(* IEC 61131-3 sources: AXOpen/src/abstractions/ctrl/src/Messaging, 18 files *)

(* ---- AxoConstants.st ---- *)
NAMESPACE AXOpen.Messaging
    TYPE PUBLIC
        AxoIntConstants : INT
        (
            MAX_MESSAGE_TEXT_LENGHT := 160,
			MDS_MAX_INDEX := 10
        );
    END_TYPE
END_NAMESPACE

(* ---- eAxoMessageDigestMethod.st ---- *)
NAMESPACE AXOpen.Messaging
    /// <summary>
    /// Message digest methods used to create fingerprint of a message.
    /// </summary>
    TYPE eAxoMessageDigestMethod : INT
    (
        /// <summary>
        /// Fastest method with highest probability of colisions.
        /// </summary>
        CRC8 := 8,

        /// <summary>
        /// Moderate speed method with lower probability of colisions.
        /// </summary>
        CRC16 := 16,

        /// <summary>
        /// Slowest speed method with relatively low probability of colisions.
        /// </summary>
        CRC32 := 32,

        /// <summary>
        /// Messages are not digested the repeated messages won't be filtered out.
        /// Use this option on low performance devices.
        /// </summary>
        NONE := 32767
    );
    END_TYPE
END_NAMESPACE

(* ---- IAxoMessageCategorize.st ---- *)
NAMESPACE AXOpen.Messaging
    INTERFACE IAxoMessageCategorize
		/// <summary>
        /// Categorizes and creates the message as 'debug'.
		/// </summary>
        METHOD AsDebug : IAxoMessageProperties END_METHOD

		/// <summary>
        /// Categorizes and creates the message as 'error'.
		/// </summary>
        METHOD AsError : IAxoMessageProperties END_METHOD

		/// <summary>
        /// Categorizes and creates the message as 'fatal'.
		/// </summary>
        METHOD AsFatal : IAxoMessageProperties END_METHOD

		/// <summary>
        /// Categorizes and creates the message as 'info'.
		/// </summary>
        METHOD AsInfo : IAxoMessageProperties END_METHOD

		/// <summary>
        /// Categorizes and creates the message as 'trace'.
		/// </summary>
        METHOD AsTrace : IAxoMessageProperties END_METHOD

		/// <summary>
        /// Categorizes and creates the message as 'warning'.
		/// </summary>
        METHOD AsWarning : IAxoMessageProperties END_METHOD
    END_INTERFACE
END_NAMESPACE

(* ---- IAxoMessageProperties.st ---- *)
NAMESPACE AXOpen.Messaging
    INTERFACE IAxoMessageProperties
        METHOD Pin: IAxoMessageProperties END_METHOD
        METHOD IsPinned: BOOL END_METHOD
    END_INTERFACE
END_NAMESPACE

(* ---- IAxoMessages.st ---- *)
NAMESPACE AXOpen.Messaging
    INTERFACE IAxoMessages
	    /// <summary>
		/// Adds message of 'debug' category to the message queue.
		/// </summary>
        METHOD Debug : IAxoMessageProperties
            VAR_INPUT
                /// <summary>
                /// Arbitrary message string.
                /// </summary>
                Message : STRING[AxoIntConstants#MAX_MESSAGE_TEXT_LENGHT];
            END_VAR
        END_METHOD

	    /// <summary>
		/// Adds message of 'error' category to the message queue.
		/// </summary>
        METHOD Error : IAxoMessageProperties
            VAR_INPUT
                /// <summary>
                /// Arbitrary message string.
                /// </summary>
                Message : STRING[AxoIntConstants#MAX_MESSAGE_TEXT_LENGHT];
            END_VAR
        END_METHOD

	    /// <summary>
		/// Adds message of 'information' category to the message queue.
		/// </summary>
        METHOD Info : IAxoMessageProperties
            VAR_INPUT
                /// <summary>
                /// Arbitrary message string.
                /// </summary>
                Message : STRING[AxoIntConstants#MAX_MESSAGE_TEXT_LENGHT];
            END_VAR
        END_METHOD

	    /// <summary>
		/// Adds message of 'notification' category to the message queue.
		/// </summary>
        METHOD Notify : IAxoMessageProperties
            VAR_INPUT
                /// <summary>
                /// Arbitrary message string.
                /// </summary>
                Message : STRING[AxoIntConstants#MAX_MESSAGE_TEXT_LENGHT];
            END_VAR
        END_METHOD

	    /// <summary>
		/// Adds message of 'programming error' category to the message queue.
		/// </summary>
        METHOD Programming : IAxoMessageProperties
            VAR_INPUT
                /// <summary>
                /// Arbitrary message string.
                /// </summary>
                Message : STRING[AxoIntConstants#MAX_MESSAGE_TEXT_LENGHT];
            END_VAR
        END_METHOD

	    /// <summary>
		/// Adds message of 'trace' category to the message queue.
		/// </summary>
        METHOD Trace : IAxoMessageProperties
            VAR_INPUT
                /// <summary>
                /// Arbitrary message string.
                /// </summary>
                Message : STRING[AxoIntConstants#MAX_MESSAGE_TEXT_LENGHT];
            END_VAR
        END_METHOD

	    /// <summary>
		/// Adds message of 'warning' category to the message queue.
		/// </summary>
        METHOD Warning : IAxoMessageProperties
            VAR_INPUT
                /// <summary>
                /// Arbitrary message string.
                /// </summary>
                Message : STRING[AxoIntConstants#MAX_MESSAGE_TEXT_LENGHT];
            END_VAR
        END_METHOD

        METHOD Build: IAxoMessageTextBuilder END_METHOD

        /// <summary>
		/// Adds message of given category to the message queue.
		/// </summary>
		/// <returns>Message index.</returns>
        METHOD Post  : IAxoMessageProperties
            VAR_INPUT
                /// <summary>
                /// Arbitrary message string.
                /// </summary>
                Message : STRING[AxoIntConstants#MAX_MESSAGE_TEXT_LENGHT];
                /// <summary>
                /// Message category.
                /// </summary>
                Category : eAxoMessageCategory;
            END_VAR
        END_METHOD

		/// <summary>
		/// Unpins this messenger.
		/// </summary>
        METHOD UnPin END_METHOD

    END_INTERFACE
END_NAMESPACE

(* ---- IAxoMessageTextBuilder.st ---- *)
NAMESPACE AXOpen.Messaging
    INTERFACE IAxoMessageTextBuilder
		/// <summary>
		/// Appends string to the message text.
		/// </summary>
		/// <remarks>
		/// 	<note type="warning">
		/// 		The size of the resulting string should not be more than '160' characters. The characters exceeding this size will be truncated.
		/// 	</note>
		/// </remarks>
 		METHOD Append : IAxoMessageTextBuilder VAR_INPUT Data : BOOL; END_VAR END_METHOD
		METHOD Append : IAxoMessageTextBuilder VAR_INPUT Data : BYTE; END_VAR END_METHOD
		METHOD Append : IAxoMessageTextBuilder VAR_INPUT Data : WORD; END_VAR END_METHOD
		METHOD Append : IAxoMessageTextBuilder VAR_INPUT Data : DWORD; END_VAR END_METHOD
		METHOD Append : IAxoMessageTextBuilder VAR_INPUT Data : LWORD; END_VAR END_METHOD
		METHOD Append : IAxoMessageTextBuilder VAR_INPUT Data : SINT; END_VAR END_METHOD
		METHOD Append : IAxoMessageTextBuilder VAR_INPUT Data : INT; END_VAR END_METHOD
		METHOD Append : IAxoMessageTextBuilder VAR_INPUT Data : DINT; END_VAR END_METHOD
		METHOD Append : IAxoMessageTextBuilder VAR_INPUT Data : LINT; END_VAR END_METHOD
		METHOD Append : IAxoMessageTextBuilder VAR_INPUT Data : USINT; END_VAR END_METHOD
		METHOD Append : IAxoMessageTextBuilder VAR_INPUT Data : UINT; END_VAR END_METHOD
		METHOD Append : IAxoMessageTextBuilder VAR_INPUT Data : UDINT; END_VAR END_METHOD
		METHOD Append : IAxoMessageTextBuilder VAR_INPUT Data : ULINT; END_VAR END_METHOD
		METHOD Append : IAxoMessageTextBuilder VAR_INPUT Data : REAL; END_VAR END_METHOD
		METHOD Append : IAxoMessageTextBuilder VAR_INPUT Data : LREAL; END_VAR END_METHOD
		METHOD Append : IAxoMessageTextBuilder VAR_INPUT Data : TIME; END_VAR END_METHOD
		METHOD Append : IAxoMessageTextBuilder VAR_INPUT Data : LTIME; END_VAR END_METHOD
		METHOD Append : IAxoMessageTextBuilder VAR_INPUT Data : DATE; END_VAR END_METHOD
		METHOD Append : IAxoMessageTextBuilder VAR_INPUT Data : LDATE; END_VAR END_METHOD
		METHOD Append : IAxoMessageTextBuilder VAR_INPUT Data : TIME_OF_DAY; END_VAR END_METHOD
		METHOD Append : IAxoMessageTextBuilder VAR_INPUT Data : LTIME_OF_DAY; END_VAR END_METHOD
		METHOD Append : IAxoMessageTextBuilder VAR_INPUT Data : DATE_AND_TIME; END_VAR END_METHOD
		METHOD Append : IAxoMessageTextBuilder VAR_INPUT Data : LDATE_AND_TIME; END_VAR END_METHOD
		METHOD Append : IAxoMessageTextBuilder VAR_INPUT Data : CHAR; END_VAR END_METHOD
		// METHOD Append : IAxoMessageTextBuilder VAR_INPUT Data : WCHAR; END_VAR END_METHOD
		METHOD Append : IAxoMessageTextBuilder VAR_INPUT Data : STRING[AxoIntConstants#MAX_MESSAGE_TEXT_LENGHT]; END_VAR END_METHOD
		// METHOD Append : IAxoMessageTextBuilder VAR_INPUT Data : WSTRING[IxIntConstants#MAX_MESSAGE_TEXT_LENGHT]; END_VAR END_METHOD
		/// <summary>
		/// Gets categorization methods for fluent message builder.
		/// </summary>
        METHOD As : IAxoMessageCategorize END_METHOD

		/// <summary>
		/// Initiates new message text building for this messenger in fluent-like fashion.
		/// </summary>
        METHOD Build : IAxoMessageTextBuilder END_METHOD
    END_INTERFACE
END_NAMESPACE

(* ---- IAxoMessenger.st ---- *)
NAMESPACE AXOpen.Messaging
    INTERFACE IAxoMessenger
		/// <summary>
		/// Clears the message content.
		/// <remarks>
		/// 	<note type="important">
		/// 		This method is exposed for Rpc calls, for testing purposes. Rpc calls of this method must not be used in production code
		///		</note>
		/// </remarks>
		/// </summary>
		METHOD Clear END_METHOD

		METHOD OnCondition : IAxoMessages
			VAR_INPUT
				inCondition : BOOL;
			END_VAR
		END_METHOD
    END_INTERFACE
END_NAMESPACE

(* ---- IAxoMessengerEnv.st ---- *)
NAMESPACE AXOpen.Messaging
    INTERFACE IAxoMessengerEnv
		/// <summary>
		/// Gets whether the messaging is suspended at this point in program.
		/// <para>
		/// See also <see cref="PlcDocu.TcoCore.TcoMessengerSettings.Resume()"/>
		/// </para>
		/// <para>
		/// See also <see cref="PlcDocu.TcoCore.TcoMessengerSettings.Suspend()"/>
		/// </para>
		/// <para>
		/// See also <see cref="PlcDocu.TcoCore.TcoMessengerSettings.MinLevel"/>
		/// </para>
		/// </summary>
		METHOD IsSuspended: BOOL END_METHOD
		/// <summary>
		/// Gets the message digest method.
		/// Message digest serves to fingerprint messages.
		/// </summary>
		METHOD GetMessageDigestMethod : eAxoMessageDigestMethod END_METHOD
		/// <summary>
		/// Sets the message digest method.
		/// Message digest serves to fingerprint messages.
		/// </summary>
		METHOD SetMessageDigestMethod VAR_INPUT inDigestMethod : eAxoMessageDigestMethod; END_VAR END_METHOD
		/// <summary>
		/// Gets the minimal messaging level, the objects will post only messages for the levels of this or superior severity.
		/// <para>
		/// See also <see cref="PlcDocu.TcoCore.TcoMessengerSettings.Resume()"/>
		/// </para>
		/// <para>
		/// See also <see cref="PlcDocu.TcoCore.TcoMessengerSettings.Suspend()"/>
		/// </para>
		/// <para>
		/// See also <see cref="PlcDocu.TcoCore.TcoMessengerSettings.MinLevel"/>
		/// </para>
		/// </summary>
		METHOD GetMinLevel : eAxoMessageCategory END_METHOD
		/// <summary>
		/// Sets the minimal messaging level, the objects will post only messages for the levels of this or superior severity.
		/// <para>
		/// See also <see cref="PlcDocu.TcoCore.TcoMessengerSettings.Resume()"/>
		/// </para>
		/// <para>
		/// See also <see cref="PlcDocu.TcoCore.TcoMessengerSettings.Suspend()"/>
		/// </para>
		/// <para>
		/// See also <see cref="PlcDocu.TcoCore.TcoMessengerSettings.MinLevel"/>
		/// </para>
		/// </summary>
		METHOD SetMinLevel VAR_INPUT inMessageCategory : eAxoMessageCategory; END_VAR END_METHOD
		/// <summary>
		/// Resumes messaging from the all objects of this context, when the messaging was previously suspended by ```Suspend``` method.
		/// <para>
		/// See also <see cref="PlcDocu.TcoCore.TcoMessengerSettings.Suspend()"/>
		/// </para>
		/// <para>
		/// See also <see cref="PlcDocu.TcoCore.TcoMessengerSettings.MinLevel"/>
		/// </para>
		/// </summary>
		METHOD Resume END_METHOD
		/// <summary>
		/// Suspends messaging from the all objects of this context that would occur from this point in the call tree.
		/// <para>
		/// See also <see cref="PlcDocu.TcoCore.TcoMessengerSettings.Resume()"/>
		/// </para>
		/// <para>
		/// See also <see cref="PlcDocu.TcoCore.TcoMessengerSettings.MinLevel"/>
		/// </para>
		/// </summary>
		METHOD Suspend END_METHOD
	END_INTERFACE
END_NAMESPACE

(* ---- IIxMessageCategorize.st ---- *)
NAMESPACE ix.framework.messaging
    INTERFACE IIxMessageCategorize
		/// <summary>
        /// Categorizes and creates the message as 'debug'.
		/// </summary>
        METHOD AsDebug : IIxMessageProperties END_METHOD

		/// <summary>
        /// Categorizes and creates the message as 'error'.
		/// </summary>
        METHOD AsError : IIxMessageProperties END_METHOD

		/// <summary>
        /// Categorizes and creates the message as 'fatal'.
		/// </summary>
        METHOD AsFatal : IIxMessageProperties END_METHOD

		/// <summary>
        /// Categorizes and creates the message as 'info'.
		/// </summary>
        METHOD AsInfo : IIxMessageProperties END_METHOD

		/// <summary>
        /// Categorizes and creates the message as 'trace'.
		/// </summary>
        METHOD AsTrace : IIxMessageProperties END_METHOD

		/// <summary>
        /// Categorizes and creates the message as 'warning'.
		/// </summary>
        METHOD AsWarning : IIxMessageProperties END_METHOD
    END_INTERFACE
END_NAMESPACE

(* ---- IIxMessages.st ---- *)
NAMESPACE ix.framework.messaging
    INTERFACE IIxMessages
	    /// <summary>
		/// Adds message of 'debug' category to the message queue.
		/// </summary>
        METHOD Debug : IIxMessageProperties
            VAR_INPUT
                /// <summary>
                /// Arbitrary message string.
                /// </summary>
                Message : STRING[IxIntConstants#MAX_MESSAGE_TEXT_LENGHT];
            END_VAR
        END_METHOD

	    /// <summary>
		/// Adds message of 'error' category to the message queue.
		/// </summary>
        METHOD Error : IIxMessageProperties
            VAR_INPUT
                /// <summary>
                /// Arbitrary message string.
                /// </summary>
                Message : STRING[IxIntConstants#MAX_MESSAGE_TEXT_LENGHT];
            END_VAR
        END_METHOD

	    /// <summary>
		/// Adds message of 'information' category to the message queue.
		/// </summary>
        METHOD Info : IIxMessageProperties
            VAR_INPUT
                /// <summary>
                /// Arbitrary message string.
                /// </summary>
                Message : STRING[IxIntConstants#MAX_MESSAGE_TEXT_LENGHT];
            END_VAR
        END_METHOD

	    /// <summary>
		/// Adds message of 'notification' category to the message queue.
		/// </summary>
        METHOD Notify : IIxMessageProperties
            VAR_INPUT
                /// <summary>
                /// Arbitrary message string.
                /// </summary>
                Message : STRING[IxIntConstants#MAX_MESSAGE_TEXT_LENGHT];
            END_VAR
        END_METHOD

	    /// <summary>
		/// Adds message of 'programming error' category to the message queue.
		/// </summary>
        METHOD Programming : IIxMessageProperties
            VAR_INPUT
                /// <summary>
                /// Arbitrary message string.
                /// </summary>
                Message : STRING[IxIntConstants#MAX_MESSAGE_TEXT_LENGHT];
            END_VAR
        END_METHOD

	    /// <summary>
		/// Adds message of 'trace' category to the message queue.
		/// </summary>
        METHOD Trace : IIxMessageProperties
            VAR_INPUT
                /// <summary>
                /// Arbitrary message string.
                /// </summary>
                Message : STRING[IxIntConstants#MAX_MESSAGE_TEXT_LENGHT];
            END_VAR
        END_METHOD

	    /// <summary>
		/// Adds message of 'warning' category to the message queue.
		/// </summary>
        METHOD Warning : IIxMessageProperties
            VAR_INPUT
                /// <summary>
                /// Arbitrary message string.
                /// </summary>
                Message : STRING[IxIntConstants#MAX_MESSAGE_TEXT_LENGHT];
            END_VAR
        END_METHOD

        METHOD Build: IIxMessageTextBuilder END_METHOD

        /// <summary>
		/// Adds message of given category to the message queue.
		/// </summary>
		/// <returns>Message index.</returns>
        METHOD Post  : IIxMessageProperties
            VAR_INPUT
                /// <summary>
                /// Arbitrary message string.
                /// </summary>
                Message : STRING[IxIntConstants#MAX_MESSAGE_TEXT_LENGHT];
                /// <summary>
                /// Message category.
                /// </summary>
                Category : eIxMessageCategory;
            END_VAR
        END_METHOD

		/// <summary>
		/// Unpins this messenger.
		/// </summary>
        METHOD UnPin END_METHOD

    END_INTERFACE
END_NAMESPACE

(* ---- IIxMessageTextBuilder.st ---- *)
NAMESPACE ix.framework.messaging
    INTERFACE IIxMessageTextBuilder
		/// <summary>
		/// Appends string to the message text.
		/// </summary>
		/// <remarks>
		/// 	<note type="warning">
		/// 		The size of the resulting string should not be more than '160' characters. The characters exceeding this size will be truncated.
		/// 	</note>
		/// </remarks>
 		METHOD Append : IIxMessageTextBuilder VAR_INPUT Data : BOOL; END_VAR END_METHOD
		METHOD Append : IIxMessageTextBuilder VAR_INPUT Data : BYTE; END_VAR END_METHOD
		METHOD Append : IIxMessageTextBuilder VAR_INPUT Data : WORD; END_VAR END_METHOD
		METHOD Append : IIxMessageTextBuilder VAR_INPUT Data : DWORD; END_VAR END_METHOD
		METHOD Append : IIxMessageTextBuilder VAR_INPUT Data : LWORD; END_VAR END_METHOD
		METHOD Append : IIxMessageTextBuilder VAR_INPUT Data : SINT; END_VAR END_METHOD
		METHOD Append : IIxMessageTextBuilder VAR_INPUT Data : INT; END_VAR END_METHOD
		METHOD Append : IIxMessageTextBuilder VAR_INPUT Data : DINT; END_VAR END_METHOD
		METHOD Append : IIxMessageTextBuilder VAR_INPUT Data : LINT; END_VAR END_METHOD
		METHOD Append : IIxMessageTextBuilder VAR_INPUT Data : USINT; END_VAR END_METHOD
		METHOD Append : IIxMessageTextBuilder VAR_INPUT Data : UINT; END_VAR END_METHOD
		METHOD Append : IIxMessageTextBuilder VAR_INPUT Data : UDINT; END_VAR END_METHOD
		METHOD Append : IIxMessageTextBuilder VAR_INPUT Data : ULINT; END_VAR END_METHOD
		METHOD Append : IIxMessageTextBuilder VAR_INPUT Data : REAL; END_VAR END_METHOD
		METHOD Append : IIxMessageTextBuilder VAR_INPUT Data : LREAL; END_VAR END_METHOD
		METHOD Append : IIxMessageTextBuilder VAR_INPUT Data : TIME; END_VAR END_METHOD
		METHOD Append : IIxMessageTextBuilder VAR_INPUT Data : LTIME; END_VAR END_METHOD
		METHOD Append : IIxMessageTextBuilder VAR_INPUT Data : DATE; END_VAR END_METHOD
		METHOD Append : IIxMessageTextBuilder VAR_INPUT Data : LDATE; END_VAR END_METHOD
		METHOD Append : IIxMessageTextBuilder VAR_INPUT Data : TIME_OF_DAY; END_VAR END_METHOD
		METHOD Append : IIxMessageTextBuilder VAR_INPUT Data : LTIME_OF_DAY; END_VAR END_METHOD
		METHOD Append : IIxMessageTextBuilder VAR_INPUT Data : DATE_AND_TIME; END_VAR END_METHOD
		METHOD Append : IIxMessageTextBuilder VAR_INPUT Data : LDATE_AND_TIME; END_VAR END_METHOD
		METHOD Append : IIxMessageTextBuilder VAR_INPUT Data : CHAR; END_VAR END_METHOD
		// METHOD Append : IIxMessageTextBuilder VAR_INPUT Data : WCHAR; END_VAR END_METHOD
		METHOD Append : IIxMessageTextBuilder VAR_INPUT Data : STRING[IxIntConstants#MAX_MESSAGE_TEXT_LENGHT]; END_VAR END_METHOD
		// METHOD Append : IIxMessageTextBuilder VAR_INPUT Data : WSTRING[IxIntConstants#MAX_MESSAGE_TEXT_LENGHT]; END_VAR END_METHOD
		/// <summary>
		/// Gets categorization methods for fluent message builder.
		/// </summary>
        METHOD As : IIxMessageCategorize END_METHOD

		/// <summary>
		/// Initiates new message text building for this messenger in fluent-like fashion.
		/// </summary>
        METHOD Build : IIxMessageTextBuilder END_METHOD
    END_INTERFACE
END_NAMESPACE

(* ---- IIxMessenger.st ---- *)
NAMESPACE ix.framework.messaging
    INTERFACE IIxMessenger
		/// <summary>
		/// Clears the message content.
		/// <remarks>
		/// 	<note type="important">
		/// 		This method is exposed for Rpc calls, for testing purposes. Rpc calls of this method must not be used in production code
		///		</note>
		/// </remarks>
		/// </summary>
		METHOD Clear END_METHOD

		METHOD OnCondition : IIxMessages
			VAR_INPUT
				inCondition : BOOL;
			END_VAR
		END_METHOD
    END_INTERFACE
END_NAMESPACE

(* ---- IIxMessengerEnv.st ---- *)
NAMESPACE ix.framework.messaging
    INTERFACE IIxMessengerEnv
		/// <summary>
		/// Gets whether the messaging is suspended at this point in program.
		/// <para>
		/// See also <see cref="PlcDocu.TcoCore.TcoMessengerSettings.Resume()"/>
		/// </para>
		/// <para>
		/// See also <see cref="PlcDocu.TcoCore.TcoMessengerSettings.Suspend()"/>
		/// </para>
		/// <para>
		/// See also <see cref="PlcDocu.TcoCore.TcoMessengerSettings.MinLevel"/>
		/// </para>
		/// </summary>
		METHOD IsSuspended: BOOL END_METHOD
		/// <summary>
		/// Gets the message digest method.
		/// Message digest serves to fingerprint messages.
		/// </summary>
		METHOD GetMessageDigestMethod : eIxMessageDigestMethod END_METHOD
		/// <summary>
		/// Sets the message digest method.
		/// Message digest serves to fingerprint messages.
		/// </summary>
		METHOD SetMessageDigestMethod VAR_INPUT inDigestMethod : eIxMessageDigestMethod; END_VAR END_METHOD
		/// <summary>
		/// Gets the minimal messaging level, the objects will post only messages for the levels of this or superior severity.
		/// <para>
		/// See also <see cref="PlcDocu.TcoCore.TcoMessengerSettings.Resume()"/>
		/// </para>
		/// <para>
		/// See also <see cref="PlcDocu.TcoCore.TcoMessengerSettings.Suspend()"/>
		/// </para>
		/// <para>
		/// See also <see cref="PlcDocu.TcoCore.TcoMessengerSettings.MinLevel"/>
		/// </para>
		/// </summary>
		METHOD GetMinLevel : eIxMessageCategory END_METHOD
		/// <summary>
		/// Sets the minimal messaging level, the objects will post only messages for the levels of this or superior severity.
		/// <para>
		/// See also <see cref="PlcDocu.TcoCore.TcoMessengerSettings.Resume()"/>
		/// </para>
		/// <para>
		/// See also <see cref="PlcDocu.TcoCore.TcoMessengerSettings.Suspend()"/>
		/// </para>
		/// <para>
		/// See also <see cref="PlcDocu.TcoCore.TcoMessengerSettings.MinLevel"/>
		/// </para>
		/// </summary>
		METHOD SetMinLevel VAR_INPUT inMessageCategory : eIxMessageCategory; END_VAR END_METHOD
		/// <summary>
		/// Resumes messaging from the all objects of this context, when the messaging was previously suspended by ```Suspend``` method.
		/// <para>
		/// See also <see cref="PlcDocu.TcoCore.TcoMessengerSettings.Suspend()"/>
		/// </para>
		/// <para>
		/// See also <see cref="PlcDocu.TcoCore.TcoMessengerSettings.MinLevel"/>
		/// </para>
		/// </summary>
		METHOD Resume END_METHOD
		/// <summary>
		/// Suspends messaging from the all objects of this context that would occur from this point in the call tree.
		/// <para>
		/// See also <see cref="PlcDocu.TcoCore.TcoMessengerSettings.Resume()"/>
		/// </para>
		/// <para>
		/// See also <see cref="PlcDocu.TcoCore.TcoMessengerSettings.MinLevel"/>
		/// </para>
		/// </summary>
		METHOD Suspend END_METHOD
	END_INTERFACE
END_NAMESPACE

(* ---- AxoMessageDigest.st ---- *)
NAMESPACE AXOpen.Messaging
    CLASS PUBLIC AxoMessageDigest
        VAR PUBLIC
            Digest : DWORD;
            Cycle : ULINT;
            Count : ULINT;
            Category : eAxoMessageCategory;
        END_VAR
    END_CLASS
END_NAMESPACE

(* ---- AxoMessengerEnv.st ---- *)
USING AXOpen.Utils;

NAMESPACE AXOpen.Messaging
    CLASS PUBLIC AxoMessengerEnv IMPLEMENTS IAxoMessengerEnv
		VAR
			_minLevel : eAxoMessageCategory;
			_isMessagingSuspended : BOOL;
			_messageDigestMethod : eAxoMessageDigestMethod := eAxoMessageDigestMethod#CRC16;
			//_messengerLoggingMethod : eIxMessengerLogMethod := eIxMessengerLogMethod#OnEventRisen;
			_sb : REF_TO AxoStringBuilder;
		END_VAR

		/// <inheritdoc />
		METHOD PUBLIC IsSuspended: BOOL
			IsSuspended := _isMessagingSuspended;
		END_METHOD

		/// <inheritdoc />
		METHOD PUBLIC GetMessageDigestMethod : eAxoMessageDigestMethod
			GetMessageDigestMethod := _messageDigestMethod;
		END_METHOD

		/// <inheritdoc />
		METHOD PUBLIC SetMessageDigestMethod
			VAR_INPUT
				inDigestMethod : eAxoMessageDigestMethod;
			END_VAR
			_messageDigestMethod := inDigestMethod;
		END_METHOD

		/// <inheritdoc />
		METHOD PUBLIC GetMinLevel : eAxoMessageCategory
			GetMinLevel := _minLevel;
		END_METHOD

		/// <inheritdoc />
		METHOD PUBLIC SetMinLevel
			VAR_INPUT
				inMessageCategory : eAxoMessageCategory;
			END_VAR
			_minLevel := inMessageCategory;
		END_METHOD

		/// <inheritdoc />
		METHOD PUBLIC Resume
			_isMessagingSuspended := FALSE;
		END_METHOD

		/// <inheritdoc />
		METHOD PUBLIC Suspend
			_isMessagingSuspended := TRUE;
		END_METHOD

		/// <inheritdoc />
		METHOD PUBLIC GetStringBuilder : REF_TO AxoStringBuilder
			GetStringBuilder ?= _sb;
		END_METHOD
	END_CLASS
END_NAMESPACE

(* ---- IxMessengerEnv.st ---- *)
USING ix.framework.utils;

NAMESPACE ix.framework.messaging
    CLASS PUBLIC IxMessengerEnv IMPLEMENTS IIxMessengerEnv
		VAR
			_minLevel : eIxMessageCategory;
			_isMessagingSuspended : BOOL;
			_messageDigestMethod : eIxMessageDigestMethod := eIxMessageDigestMethod#CRC16;
			//_messengerLoggingMethod : eIxMessengerLogMethod := eIxMessengerLogMethod#OnEventRisen;
			_sb : REF_TO StringBuilder;
		END_VAR

		/// <inheritdoc />
		METHOD PUBLIC IsSuspended: BOOL
			IsSuspended := _isMessagingSuspended;
		END_METHOD

		/// <inheritdoc />
		METHOD PUBLIC GetMessageDigestMethod : eIxMessageDigestMethod
			GetMessageDigestMethod := _messageDigestMethod;
		END_METHOD

		/// <inheritdoc />
		METHOD PUBLIC SetMessageDigestMethod
			VAR_INPUT
				inDigestMethod : eIxMessageDigestMethod;
			END_VAR
			_messageDigestMethod := inDigestMethod;
		END_METHOD

		/// <inheritdoc />
		METHOD PUBLIC GetMinLevel : eIxMessageCategory
			GetMinLevel := _minLevel;
		END_METHOD

		/// <inheritdoc />
		METHOD PUBLIC SetMinLevel
			VAR_INPUT
				inMessageCategory : eIxMessageCategory;
			END_VAR
			_minLevel := inMessageCategory;
		END_METHOD

		/// <inheritdoc />
		METHOD PUBLIC Resume
			_isMessagingSuspended := FALSE;
		END_METHOD

		/// <inheritdoc />
		METHOD PUBLIC Suspend
			_isMessagingSuspended := TRUE;
		END_METHOD

		/// <inheritdoc />
		METHOD PUBLIC GetStringBuilder : REF_TO StringBuilder
			GetStringBuilder ?= _sb;
		END_METHOD
	END_CLASS
END_NAMESPACE

(* ---- eAxoMessageCategory.st ---- *)
NAMESPACE AXOpen.Messaging
    TYPE PUBLIC
        ///<summary>
        /// Message categories.
        /// ATTENTION: Values must be multiply of 100
        ///</summary>
        eAxoMessageCategory : INT
        (
            All := 0,

            ///<summary>
            /// Trace message to be used for tracing purpose.
            /// Use when you need to track detailed information about internal states of the program for detailed visibility.
            /// This is lowest level of category that can be used in production, for detailed observation of PLC program.
            ///</summary>
            Trace := 100,

            ///<summary>
            /// Debug message to be used for debugging purpose only.
            /// Use when you need to report debug information for you as programmer.
            ///</summary>
            Debug := 200,

            ///<summary>
            /// Info message.
            /// Use when you want to deliver information to the user, that has only informative character and does not adversely affect a process.
            ///</summary>
            Info := 300,

            ///<summary>
            /// Time-out message.
            /// Use this category when you want to report a timed-out information, that may eventually succed.
            ///</summary>
            TimedOut := 400,

            ///<summary>
            /// Notification message.
            /// Use this category when you want to report a notification that may be of interest to the user, but does not adversly affect a process.
            ///</summary>
            Notification := 500,

            ///<summary>
            /// Warning message.
            /// Use this category when you want to report to the user an information about a possible problem, that may adversly affect a process.
            /// Information in this cateogory aims to help the user to identify a problem, the cause of such problem does not necessarily stops the process.
            ///</summary>
            Warning := 600,

            ///<summary>
            /// Error message.
            /// Use this categoty when there is a failure that cannot be immediately recovered and an intervention is needed. This is typically a situation when a device fails
            /// to deliver expected result.
            /// Do not use this category to report information about failed process like measurement or detection.
            ///</summary>
            Error := 700,

            ///<summary>
            /// Programming issue.
            /// Use this category to inform about a possible programming error, defect in settings or missing information at a level of programming or system or process settings.
            ///</summary>
            ProgrammingError := 900,

            ///<summary>
            /// Critical error.
            /// Use this category when a critical error occured, that is not recoverable by the means of software (reset/restore) but device still operates under such conditions; a detailed inspection and an expert action is required.
            ///</summary>
            Critical := 1000,

            ///<summary>
            /// Fatal error.
            /// Use this category when a fatal error occured, that is not recoverable by the means of software (reset/restore) and a detailed inspection is required, the device is not able to continue without special intervention,
            ///</summary>
            Fatal    := 1100,

            ///<summary>
            /// Catastrophic error.
            /// Use this category when there is a situation when the device cannot continue operations due to irrecoverable failure.
            ///</summary>
            Catastrophic := 1200,

            None := 32000
        );
    END_TYPE
END_NAMESPACE

(* ---- eIxMessageCategory.st ---- *)
NAMESPACE ix.framework.messaging
    TYPE PUBLIC
        ///<summary>
        /// Message categories.
        /// ATTENTION: Values must be multiply of 100
        ///</summary>
        eIxMessageCategory : INT
        (
            All := 0,

            ///<summary>
            /// Trace message to be used for tracing purpose.
            /// Use when you need to track detailed information about internal states of the program for detailed visibility.
            /// This is lowest level of category that can be used in production, for detailed observation of PLC program.
            ///</summary>
            Trace := 100,

            ///<summary>
            /// Debug message to be used for debugging purpose only.
            /// Use when you need to report debug information for you as programmer.
            ///</summary>
            Debug := 200,

            ///<summary>
            /// Info message.
            /// Use when you want to deliver information to the user, that has only informative character and does not adversely affect a process.
            ///</summary>
            Info := 300,

            ///<summary>
            /// Time-out message.
            /// Use this category when you want to report a timed-out information, that may eventually succed.
            ///</summary>
            TimedOut := 400,

            ///<summary>
            /// Notification message.
            /// Use this category when you want to report a notification that may be of interest to the user, but does not adversly affect a process.
            ///</summary>
            Notification := 500,

            ///<summary>
            /// Warning message.
            /// Use this category when you want to report to the user an information about a possible problem, that may adversly affect a process.
            /// Information in this cateogory aims to help the user to identify a problem, the cause of such problem does not necessarily stops the process.
            ///</summary>
            Warning := 600,

            ///<summary>
            /// Error message.
            /// Use this categoty when there is a failure that cannot be immediately recovered and an intervention is needed. This is typically a situation when a device fails
            /// to deliver expected result.
            /// Do not use this category to report information about failed process like measurement or detection.
            ///</summary>
            Error := 700,

            ///<summary>
            /// Programming issue.
            /// Use this category to inform about a possible programming error, defect in settings or missing information at a level of programming or system or process settings.
            ///</summary>
            ProgrammingError := 900,

            ///<summary>
            /// Critical error.
            /// Use this category when a critical error occured, that is not recoverable by the means of software (reset/restore) but device still operates under such conditions; a detailed inspection and an expert action is required.
            ///</summary>
            Critical := 1000,

            ///<summary>
            /// Fatal error.
            /// Use this category when a fatal error occured, that is not recoverable by the means of software (reset/restore) and a detailed inspection is required, the device is not able to continue without special intervention,
            ///</summary>
            Fatal    := 1100,

            ///<summary>
            /// Catastrophic error.
            /// Use this category when there is a situation when the device cannot continue operations due to irrecoverable failure.
            ///</summary>
            Catastrophic := 1200,

            None := 32000
        );
    END_TYPE
END_NAMESPACE
